INTERFACE I_Command

METHOD Execute
VAR_INPUT
END_VAR
END_METHOD

END_INTERFACE

(* stored: Version 1.1.0.1, ProductVersion 3.1.4024.11
   Itf I_Command: Id {def6fb86-9ebc-4ca3-ad88-695ce27a42b2}
   Method Execute: Id {d830acd0-c431-4de1-beff-f8f4f750a898} *)
